FUNCTION_BLOCK FB_SLITS_POWER EXTENDS FB_SLITS
VAR_INPUT
END_VAR
VAR
     {attribute 'pytmc' := '
        pv: FSW
    '}
    fbFlowSwitch: FB_XTES_Flowswitch;


    //RTDs
    {attribute 'pytmc' := '
        pv: TOP:RTD:01
    '}
    RTD_TOP_1: FB_TempSensor;
    {attribute 'pytmc' := '
        pv: TOP:RTD:02
    '}
    RTD_TOP_2: FB_TempSensor;
    {attribute 'pytmc' := '
        pv: BOTTOM:RTD:01
    '}
    RTD_Bottom_1: FB_TempSensor;
    {attribute 'pytmc' := '
        pv: BOTTOM:RTD:02
    '}
    RTD_Bottom_2: FB_TempSensor;

    {attribute 'pytmc' := '
        pv: NORTH:RTD:01
    '}
    RTD_North_1: FB_TempSensor;
    {attribute 'pytmc' := '
        pv: NORTH:RTD:02
    '}
    RTD_North_2: FB_TempSensor;
    {attribute 'pytmc' := '
        pv: SOUTH:RTD:01
    '}
    RTD_South_1: FB_TempSensor;
    {attribute 'pytmc' := '
        pv: SOUTH:RTD:02
    '}
    RTD_South_2: FB_TempSensor;


END_VAR


ACT_RTDs();

ACTION ACT_RTDs:
////RTDs
RTD_TOP_1();
RTD_TOP_2();
RTD_Bottom_1();
RTD_Bottom_2();
RTD_North_1();
RTD_North_2();
RTD_South_1();
RTD_South_2();

//Flow Switch
fbFlowSwitch();
END_ACTION

END_FUNCTION_BLOCK

(* stored: Version 1.1.0.1, ProductVersion 3.1.4022.18
   POU FB_SLITS_POWER: Id {d889b456-91f0-0980-2255-32e7e69e3656}, SpecialFunc None
   Action ACT_RTDs: Id {2824f268-7671-0ba5-2fec-76114d5b195e} *)
